Staubli VAL3: delStrArray1.pgx

public program delStrArray1(string& x_sStrIn[], num x_nPos, num x_nNum)
  local num l_nSize
  local num l_i
begin
  //删除字符串数组
  //x_sStrIn:返回的新数组
  //x_nPos：起始位置
  //x_nNum:删除数组个数
  //取整
  x_nNum=roundDown(x_nNum)
  if x_nNum<1
    return
  endIf
  if x_nNum>size(x_sStrIn)
    x_nNum=size(x_sStrIn)
  endIf

  //
  if x_nPos<0
    x_nPos=0
  else
    if x_nPos>size(x_sStrIn)-1
      x_nPos=size(x_sStrIn)-1
    endIf
  endIf
  //
  if size(x_sStrIn)<=1
    x_sStrIn=""
    return
  endIf
  //
  for l_i=x_nPos to min(size(x_sStrIn)-1,x_nPos+x_nNum-1)
    delete(x_sStrIn[size(x_sStrIn)-1])
  endFor
end
